TYPE ST_HMI_Monitor_AcDcCharger :
STRUCT
	state 			: STRING;
	available 		: BOOL;
	r_AcCurrentMax	: REAL;
	r_AcPowerMax	: REAL;
	r_DcPower 		: REAL;
	r_AcPower 		: REAL;
	r_AcCurrent		: REAL;
	r_AcVoltage		: REAL;
END_STRUCT
END_TYPE

(* stored: Version 1.1.0.1, ProductVersion 3.1.4026.18
   DUT ST_HMI_Monitor_AcDcCharger: Id {4fd508a2-30dc-4c1c-94dc-380e67802db8} *)
